PROGRAM MAIN
VAR
END_VAR

END_PROGRAM

(* stored: Version 1.1.0.1
   POU MAIN: Id {42ad8e47-654e-42ec-ae6b-6940aa65046f} *)
